/// Turck RFID IO structure.
TYPE ST_FurnaceIO :
STRUCT
	
	/// Data to device.           
	stOut		AT%Q*		: ST_FurnaceOut;
	
	/// Data from device.
	stIn		AT%I*		: ST_FurnaceIn;
	
END_STRUCT
END_TYPE

(* stored: Version 1.1.0.1
   DUT ST_FurnaceIO: Id {1e20d351-cebc-4dda-a3ab-1c7c5f750142} *)
